FUNCTION putUsint : BOOL
	VAR_INPUT
		usintVar : USINT;
	END_VAR
	VAR_IN_OUT
		bufferRef : POINTER TO USINT;
	END_VAR

	memcpy(bufferRef, ADR(usintVar), SIZEOF(USINT));
	bufferRef := bufferRef + SIZEOF(USINT);
	putUsint := TRUE;

END_FUNCTION

(* stored: Version 1.1.0.1, ProductVersion 3.1.4024.3
   POU putUsint: Id {81d3eaa4-5932-00bf-2b34-50c4bfff61c5}, SpecialFunc None *)
